// TwinCAT 3 PLC project ADS_PLC
// ProgramVersion: 3.1.4023.0
// libraries:
//   Tc2_Standard, * (Beckhoff Automation GmbH)
//   Tc2_System, * (Beckhoff Automation GmbH)
//   Tc3_Module, * (Beckhoff Automation GmbH)
// project tree:
//   DUTs/ E_METHOD.TcDUT, E_OPERATION.TcTLEO, ST_CAT.TcDUT, ST_HEADER_FIELDS.TcDUT, ST_HTTP_MESSAGE.TcDUT, ST_MESSAGE_INFO.TcDUT, ST_REQUEST_LINE.TcDUT, ST_STRUCT.TcDUT
//   / PlcTask.TcTTO
//   POUs/ FB_Messenger.TcPOU, MAIN.TcPOU
// real-time tasks:
//   TASK PlcTask: cycle T#1ms, priority 20, ADS port 350

CONFIGURATION ADS_PLC
    RESOURCE PLC ON TwinCAT3
        TASK PlcTask(INTERVAL := T#1ms, PRIORITY := 20);
        PROGRAM MAIN WITH PlcTask : MAIN;
    END_RESOURCE
END_CONFIGURATION

// ---- DUTs/E_METHOD.TcDUT
{attribute 'qualified_only'}
{attribute 'strict'}
TYPE E_METHOD :
(
	GET := 0,
	HEAD,
	POST,
	PUT,
	DELETE,
	CONNECT,
	OPTIONS
)UINT;
END_TYPE

// ---- DUTs/E_OPERATION.TcTLEO
{attribute 'qualified_only'}
{attribute 'strict'}
TYPE E_OPERATION :
(
	Array_Sum 	:= 0,
	Array_Product
);
END_TYPE

// ---- DUTs/ST_CAT.TcDUT
TYPE ST_CAT :
STRUCT
	bValue0, 
	bValue1 : BOOL;
	fValue 	: REAL; 
END_STRUCT
END_TYPE

// ---- DUTs/ST_HEADER_FIELDS.TcDUT
TYPE ST_HEADER_FIELDS :
STRUCT
	sHost,
	sAccept, 
	sAccept_Language,
	sAccept_Encoding,
	sUser_Agent 		: T_MaxString;
END_STRUCT
END_TYPE

// ---- DUTs/ST_HTTP_MESSAGE.TcDUT
TYPE ST_HTTP_MESSAGE :
STRUCT
	stRequest_Line : ST_REQUEST_LINE;
	stHeader_Fields : ST_HEADER_FIELDS;
END_STRUCT
END_TYPE

// ---- DUTs/ST_MESSAGE_INFO.TcDUT
TYPE ST_MESSAGE_INFO :
STRUCT
	tTimestamp 	 : DT;
	sDescription : T_MaxString;
	eOperation 	 : E_OPERATION;
END_STRUCT
END_TYPE

// ---- DUTs/ST_REQUEST_LINE.TcDUT
TYPE ST_REQUEST_LINE :
STRUCT
	eMethod 	: E_METHOD;
	sURI 		: T_MaxString;
	sProtocol 	: T_MaxString;
END_STRUCT
END_TYPE

// ---- DUTs/ST_STRUCT.TcDUT
TYPE ST_STRUCT :
STRUCT
	bValue : BOOL;
	tTimestamp : DT;
	fValue : LREAL;
END_STRUCT
END_TYPE

// ---- POUs/MAIN.TcPOU
PROGRAM MAIN
VAR
	fbMessanger 			: FB_Messenger;
	arstHTTP_Messages_In 	: ARRAY[0..2] OF ST_HTTP_MESSAGE;
	arstHTTP_Messages_Out 	: ARRAY[0..2] OF ST_HTTP_MESSAGE;
	arstStruct 				: ARRAY [0..999] OF ST_STRUCT;
	arstCat 				: ARRAY [0..99] OF ST_CAT;
END_VAR
VAR CONSTANT
	arstRequest_Line : ARRAY[0..2] OF ST_REQUEST_LINE :=
									[ 
										( eMethod := E_METHOD.GET, sURI := '/brands/toyota.html', sProtocol := 'HTTP/1.1'),
										( eMethod := E_METHOD.GET, sURI := '/brands/suzuki.html', sProtocol := 'HTTP/1.1'),
										( eMethod := E_METHOD.GET, sURI := '/_/mss/boq-one-google/_/js', sProtocol := 'HTTP/1.1')
									];
	arstHeader_Fields : ARRAY[0..2] OF ST_HEADER_FIELDS := 
									[
										(sHost := 'www.cars.com', sAccept := 'text/html text/plain image/gif image/jpeg', sAccept_Language := 'en-GB', sAccept_Encoding := 'gzip, deflate', sUser_Agent := 'Safari/537.36'),
										(sHost := 'www.cars.com', sAccept := 'text/html text/plain image/gif image/jpeg', sAccept_Language := 'en-US,en;q=0.9', sAccept_Encoding := 'gzip, deflate', sUser_Agent := 'Chrome/102.0.5005.124'),
										(sHost := 'www.gstatic.com', sAccept := '*/*', sAccept_Language := 'en-US,en;q=0.9', sAccept_Encoding := 'gzip, deflate, br', sUser_Agent := 'Mozilla/5.0')
									];
END_VAR

arstHTTP_Messages_Out[0].stRequest_Line := arstRequest_Line[0];
arstHTTP_Messages_Out[0].stHeader_Fields := arstHeader_Fields[0];

arstHTTP_Messages_Out[1].stRequest_Line := arstRequest_Line[1];
arstHTTP_Messages_Out[1].stHeader_Fields := arstHeader_Fields[1];

arstHTTP_Messages_Out[2].stRequest_Line := arstRequest_Line[2];
arstHTTP_Messages_Out[2].stHeader_Fields := arstHeader_Fields[2];

END_PROGRAM

// ---- POUs/FB_Messenger.TcPOU
FUNCTION_BLOCK FB_Messenger
VAR_INPUT
END_VAR
VAR_OUTPUT
END_VAR
VAR
END_VAR

{attribute 'TcRpcEnable'}
METHOD Send : LREAL
VAR_INPUT
	stMessage_Info 	: ST_MESSAGE_INFO;
	arfData 		: ARRAY[0..2] OF LREAL;
END_VAR
VAR_OUTPUT
	sReturn_Message : WSTRING;
	bSuccess 		: BOOL; 
END_VAR
VAR_INST 
	stMessage_Info_Copy : ST_MESSAGE_INFO;
	arfData_Copy : ARRAY[0..2] OF LREAL;
END_VAR
VAR 
	i : DINT;
END_VAR
stMessage_Info_Copy := stMessage_Info;
arfData_Copy 		:= arfData;

CASE stMessage_Info.eOperation OF
	E_OPERATION.Array_Sum:
		FOR i := 0 TO SIZEOF(arfDATA)/SIZEOF(arfData[0])-1 DO
			Send := Send + arfData[i];
			END_FOR
	E_OPERATION.Array_Product:
		Send := arfData[0];
		FOR i := 1 TO SIZEOF(arfDATA)/SIZEOF(arfData[0])-1 DO
			Send := Send * arfData[i];
			END_FOR
END_CASE

sReturn_Message := "I have finished!";
bSuccess 		:= TRUE;
END_METHOD

END_FUNCTION_BLOCK
